FUNCTION TryConvert_USINT_TO_LWORD : BOOL
VAR_INPUT
	in : USINT;
	out : REFERENCE TO LWORD;
END_VAR

out := USINT_TO_LWORD(in);
TryConvert_USINT_TO_LWORD := TRUE;

END_FUNCTION

(* stored: Version 1.1.0.1, ProductVersion 3.1.4024.12
   POU TryConvert_USINT_TO_LWORD: Id {c3961fac-23fc-4dd3-91a1-dd8eb41d8eab}, SpecialFunc None *)
